(* PLC project Unnamed, Unknown Unnamed 1 *)
(* stored: creationDateTime 2025-06-13T16:30:15, modificationDateTime 2025-06-13T17:08:17 *)

PROGRAM part3
  VAR
    state : UINT := 0;
    wait_for_request : UINT := 0;
    wait_for_traffic : UINT := 1;
    slow_cars : UINT := 2;
    ped_xing : UINT := 3;
    all_red : UINT := 4;
  END_VAR
  VAR
    car_sensor AT %IX0.0 : BOOL;
    ped_button AT %IX0.1 : BOOL;
    car_red AT %QX0.0 : BOOL;
    car_yellow AT %QX0.1 : BOOL;
    car_green AT %QX0.2 : BOOL;
    ped_red AT %QX0.3 : BOOL;
    ped_green AT %QX0.4 : BOOL;
  END_VAR
  VAR
    TON0 : TON;
    yellow_delay : TIME := T#3s;
    ped_xing_delay : TIME := T#15s;
    all_red_delay : TIME := T#1s;
    TON1 : TON;
    TON2 : TON;
  END_VAR
  VAR  (* added by the conversion: wires and edge detectors of the diagram *)
    _EQ1_OUT : BOOL;
    _EQ4_OUT : BOOL;
    _EQ7_OUT : BOOL;
    _EQ10_OUT : BOOL;
    _EQ13_OUT : BOOL;
  END_VAR

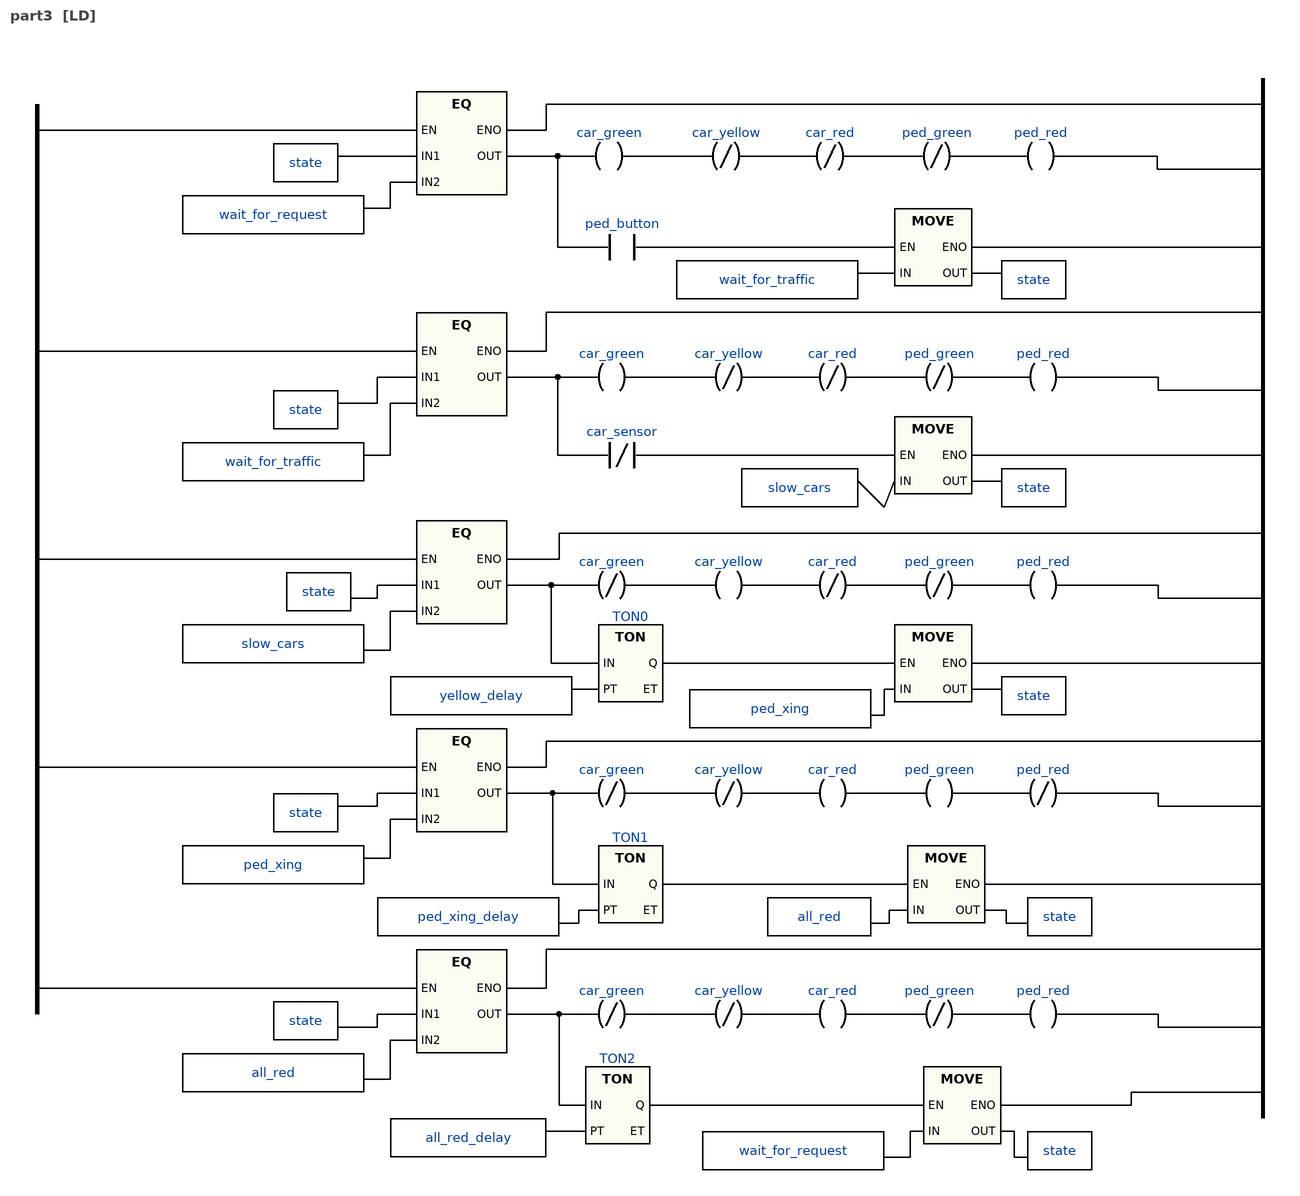
(* LD diagram, written out as Structured Text *)
_EQ1_OUT := state = wait_for_request;
car_green := _EQ1_OUT;
ped_red := _EQ1_OUT;
ped_green := NOT _EQ1_OUT;
car_yellow := NOT _EQ1_OUT;
car_red := NOT _EQ1_OUT;
_EQ4_OUT := state = wait_for_traffic;
car_green := _EQ4_OUT;
ped_red := _EQ4_OUT;
ped_green := NOT _EQ4_OUT;
car_yellow := NOT _EQ4_OUT;
car_red := NOT _EQ4_OUT;
_EQ7_OUT := state = slow_cars;
car_green := NOT _EQ7_OUT;
ped_red := _EQ7_OUT;
ped_green := NOT _EQ7_OUT;
car_yellow := _EQ7_OUT;
car_red := NOT _EQ7_OUT;
_EQ10_OUT := state = ped_xing;
car_green := NOT _EQ10_OUT;
ped_red := NOT _EQ10_OUT;
ped_green := _EQ10_OUT;
car_yellow := NOT _EQ10_OUT;
car_red := _EQ10_OUT;
_EQ13_OUT := state = all_red;
car_green := NOT _EQ13_OUT;
ped_red := _EQ13_OUT;
ped_green := NOT _EQ13_OUT;
car_yellow := NOT _EQ13_OUT;
car_red := _EQ13_OUT;
IF _EQ1_OUT AND ped_button THEN state := wait_for_traffic; END_IF;
IF _EQ4_OUT AND NOT car_sensor THEN state := slow_cars; END_IF;
TON0(IN := _EQ7_OUT, PT := yellow_delay);
IF TON0.Q THEN state := ped_xing; END_IF;
TON1(IN := _EQ10_OUT, PT := ped_xing_delay);
IF TON1.Q THEN state := all_red; END_IF;
TON2(IN := _EQ13_OUT, PT := all_red_delay);
IF TON2.Q THEN state := wait_for_request; END_IF;
END_PROGRAM

CONFIGURATION Config0
  RESOURCE Res0 ON PLC
    TASK task0(INTERVAL := T#20ms, PRIORITY := 0);
    PROGRAM instance0 WITH task0 : part3;
  END_RESOURCE
END_CONFIGURATION
